INTERFACE PUBLIC I_Command EXTENDS Disposable

METHOD PUBLIC Execute
END_METHOD

END_INTERFACE

(* stored: Version 1.1.0.1
   Itf I_Command: Id {5482795c-4fc0-4be1-b623-899f29e63002}
   Method Execute: Id {cd320ce1-cc3a-4e76-811c-b70da7184772} *)
